TYPE ST_DiagMessage :
STRUCT
	nDiagCode: UDINT;
	nFlags: ST_DiagMessageFlags;
	/// The text defined in the ESI file (//DiagMessages)
	nTextID: UINT;
	nTimeStamp: ULINT;
	aParameter: ARRAY[1..16] OF BYTE;
END_STRUCT
END_TYPE

(* stored: Version 1.1.0.1, ProductVersion 3.1.4024.12
   DUT ST_DiagMessage: Id {50aa2c0d-1f9c-4898-8fba-d772dd37fb94} *)
